(* IEC 61131-3 sources: volt/packages/volt-lsp-iec/test-corpus/pro2193/Device/Plc Logic/Application/09 Misc/Library Manager/CmpDynamicText, 18 files *)

(* ---- SVN_INFO_FLAGS.gvl ---- *)
VAR_GLOBAL
	XINCOMPLETE : BOOL := FALSE;
	XMODIFIED : BOOL := TRUE;
	XSWITCHED : BOOL := FALSE;
	XCLEAN : BOOL := FALSE;
	XDISCONNECTED : BOOL := FALSE;
END_VAR

(* ---- SVN_INFO_LASTCHANGE.gvl ---- *)
VAR_GLOBAL
	DTLASTCHANGEUTC : DATE_AND_TIME := DATE_AND_TIME#2021-2-4-15:22:35;
	WSLASTCHANGELOCAL : WSTRING(44) := "2021-02-04 16:22:35 +0100 (Thu, 04 Feb 2021)";
	WSLASTCHANGEAUTHOR : WSTRING(8) := "b.schurr";
END_VAR

(* ---- SVN_INFO_REVISIONS.gvl ---- *)
VAR_GLOBAL
	LIMINREVISION : LINT := LINT#52494;
	LIMAXREVISION : LINT := LINT#52494;
END_VAR

(* ---- SVN_INFO_SUMMARY.gvl ---- *)
VAR_GLOBAL
	SVERSIONSUMMARY : STRING(6) := '52494M';
END_VAR

(* ---- SVN_INFO_SUMMARYW.gvl ---- *)
VAR_GLOBAL
	WSVERSIONSUMMARY : WSTRING(6) := "52494M";
END_VAR

(* ---- SVN_INFO_URI.gvl ---- *)
VAR_GLOBAL
	WURL : WSTRING(97) := "svn://server04/LibrariesV3Source/branches/V3.5.17.0/System/SysLibs/CmpDynamicText/CmpDynamicText/";
END_VAR

(* ---- DYNAMICTEXTCHANGELANGUAGE.pou ---- *)
FUNCTION DYNAMICTEXTCHANGELANGUAGE : BOOL
VAR_INPUT
	STLANGUAGE : STRING;
END_VAR
END_FUNCTION

(* ---- DYNAMICTEXTGETCURRENTLANGUAGE.pou ---- *)
FUNCTION DYNAMICTEXTGETCURRENTLANGUAGE : STRING
END_FUNCTION

(* ---- DYNAMICTEXTGETDEFAULTTEXT.pou ---- *)
FUNCTION DYNAMICTEXTGETDEFAULTTEXT : POINTER TO STRING
VAR_INPUT
	PSTTEXTLIST : POINTER TO STRING;
	PSTTEXTINDEX : POINTER TO STRING;
END_VAR
END_FUNCTION

(* ---- DYNAMICTEXTGETDEFAULTTEXTW.pou ---- *)
FUNCTION DYNAMICTEXTGETDEFAULTTEXTW : POINTER TO STRING
VAR_INPUT
	PSTTEXTLIST : POINTER TO STRING;
	PSTTEXTINDEX : POINTER TO STRING;
END_VAR
END_FUNCTION

(* ---- DYNAMICTEXTGETTEXT.pou ---- *)
FUNCTION DYNAMICTEXTGETTEXT : POINTER TO STRING
VAR_INPUT
	PSTTEXTLIST : POINTER TO STRING;
	PSTTEXTINDEX : POINTER TO STRING;
END_VAR
END_FUNCTION

(* ---- DYNAMICTEXTGETTEXTW.pou ---- *)
FUNCTION DYNAMICTEXTGETTEXTW : POINTER TO STRING
VAR_INPUT
	PSTTEXTLIST : POINTER TO STRING;
	PSTTEXTINDEX : POINTER TO STRING;
END_VAR
END_FUNCTION

(* ---- DYNAMICTEXTITERATEINDICES.pou ---- *)
FUNCTION DYNAMICTEXTITERATEINDICES : RTS_IEC_RESULT
VAR_INPUT
	PSTTEXTLIST : POINTER TO STRING;
	PFITERATIONCALLBACK : POINTER TO BYTE;
	ITERATIONDATA : __UXINT;
END_VAR
END_FUNCTION

(* ---- DYNAMICTEXTLOADDEFAULTTEXTS.pou ---- *)
FUNCTION DYNAMICTEXTLOADDEFAULTTEXTS : RTS_IEC_RESULT
END_FUNCTION

(* ---- DYNAMICTEXTREGISTERFILE.pou ---- *)
FUNCTION DYNAMICTEXTREGISTERFILE : RTS_IEC_RESULT
VAR_INPUT
	SZFILE : REFERENCE TO STRING;
END_VAR
END_FUNCTION

(* ---- DYNAMICTEXTREGISTERPATH.pou ---- *)
FUNCTION DYNAMICTEXTREGISTERPATH : RTS_IEC_RESULT
VAR_INPUT
	SZPATH : REFERENCE TO STRING;
END_VAR
END_FUNCTION

(* ---- DYNAMICTEXTRELOADTEXTS.pou ---- *)
FUNCTION DYNAMICTEXTRELOADTEXTS : RTS_IEC_RESULT
END_FUNCTION

(* ---- DYNAMICTEXTUNREGISTERFILE.pou ---- *)
FUNCTION DYNAMICTEXTUNREGISTERFILE : RTS_IEC_RESULT
VAR_INPUT
	SZFILE : REFERENCE TO STRING;
END_VAR
END_FUNCTION
